FUNCTION_BLOCK ConveyProduct EXTENDS BaseState
VAR_INPUT
END_VAR
VAR_OUTPUT
END_VAR
VAR
END_VAR

METHOD mIrun : BOOL
BasePointer^.ConveyorAccessI[1].mAutoOn();
BasePointer^.ElevatorAccessI[1].mAutoOn();
BasePointer^.MixerAccessI[1].mAutoOn();
mNextState();
END_METHOD

END_FUNCTION_BLOCK

(* stored: Version 1.1.0.1, ProductVersion 3.1.4024.12
   POU ConveyProduct: Id {6d99734e-050e-41c2-8b96-5f9a09ed2639}, SpecialFunc None
   Method mIrun: Id {390f3587-73bf-4de4-a32b-a10269890d34} *)
